{attribute 'linkalways'} 
{attribute 'no_explicit_call' := 'This FB is a CLASS and must be accessed using methods or properties'}
{attribute 'enable_dynamic_creation'}
FUNCTION_BLOCK FINAL XOR_BOOL EXTENDS Node
VAR
	in1 : _BOOL(FALSE);
	in2 : _BOOL(FALSE);
	out : _BOOL(FALSE);
END_VAR

METHOD PUBLIC Clone : I_Node
VAR
	pNode : POINTER TO XOR_BOOL;
END_VAR
pNode := __NEW(XOR_BOOL);
Clone := pNode^;
END_METHOD

METHOD FB_init : BOOL
VAR_INPUT
	bInitRetains : BOOL; // if TRUE, the retain variables are initialized (warm start / cold start)
	bInCopyCode : BOOL;  // if TRUE, the instance afterwards gets moved into the copy code (online change)
END_VAR
AddInput('in1',THIS^.in1);
AddInput('in2',THIS^.in2);
AddOutput('out', THIS^.out);
END_METHOD

METHOD PROTECTED OnExecute
VAR
END_VAR
out.Value := in1.Value XOR in2.Value;
END_METHOD

END_FUNCTION_BLOCK

(* stored: Version 1.1.0.1, ProductVersion 3.1.4024.15
   POU XOR_BOOL: Id {f5481aec-60a4-44f2-bd14-74e936591349}, SpecialFunc None
   Folder Constructor: Id {841ad2f0-43e8-4eb8-b9aa-32ced934c773}
   Method Clone: Id {f8b05f8a-84b7-497e-9bcc-fdabde4d68f5}
   Method FB_init: Id {592d1f22-c0fe-49a9-aa8e-da04c0452b96}
   Method OnExecute: Id {422de39a-83a5-4ff2-bba9-71f00a6c626c} *)
